FUNCTION_BLOCK ha_timer (* ODE_init *)
  (* Standard: 61499-2 *)
  (* Version 0.1, 2017-00-25, hpea485, UOA *)
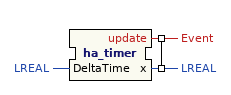
  EVENT_OUTPUT
    update WITH x;
  END_EVENT
  VAR_INPUT
    DeltaTime : LREAL := 0.01;
  END_VAR
  VAR_OUTPUT
    x : LREAL;
  END_VAR
  VAR
    Variable1 : BOOL;
  END_VAR
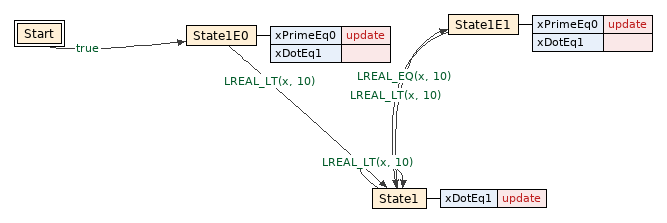
  EC_STATES
    Start;
    State1E0 : xPrimeEq0 -> update, xDotEq1;
    State1 : xDotEq1 -> update;
    State1E1 : xPrimeEq0 -> update, xDotEq1;
  END_STATES
  EC_TRANSITIONS
    Start TO State1E0 := true;
    State1E0 TO State1 := LREAL_LT(x, 10);
    State1 TO State1E1 := LREAL_EQ(x, 10);
    State1 TO State1 := LREAL_LT(x, 10);
    State1E1 TO State1 := LREAL_LT(x, 10);
  END_TRANSITIONS
  ALGORITHM xDotEq1 IN C: (* ODE *)
x_dot = 1;
  END_ALGORITHM
  ALGORITHM xPrimeEq0 IN C: (* ODE_init *)
x_prime = 0;
  END_ALGORITHM
END_FUNCTION_BLOCK
